{attribute 'qualified_only'}
TYPE e_EthercatState :
(
	Error:=0,
	INIT := 1,
	PREOP :=2,
	BOOT :=3,
	SAFEOP:=4,
	OP :=8

);
END_TYPE

(* stored: Version 1.1.0.1, ProductVersion 3.1.4024.12
   DUT e_EthercatState: Id {b30b18ec-b8cc-4149-8c7f-d5473e66c7b7} *)
